{attribute 'GeneratedUsingTerminal: ATH2000-5250-0022'}
{attribute addProperty BoxType "ATH2000-5250-0022"}
{attribute addProperty Id "BinaryDataAT %I*ARRAY [0..63] OF BYTE0"}
{attribute addProperty CRC "761682001"}
{attribute addProperty Size "0"}
TYPE FB_Inputs_2D665851 :
STRUCT
	{attribute addProperty Name "BinaryData"}
	BinaryData AT %I* : ARRAY [0..63] OF BYTE;
END_STRUCT
END_TYPE

(* stored: Version 1.2.0.0, ProductVersion 3.1.4024.9
   DUT FB_Inputs_2D665851: Id {c5d443f5-5930-44b9-962c-cdc1d37fea27} *)
